//bit packed sint;
myStopMode.0 := bNo_Ramp_Stop;
myStopMode.1 := bFollowing_Error_Stop;

//34.001  AMC Stop Mode
//AMC StopMode(34.001)
WriteUserParameterSINT(00,34,001,myStopMode);
	
//41.007  AMC Following Error Window
//Set the following error window.
IF diFollowing_Error_Window < 0 THEN
	WriteUserParameterDINT(00,41,007,0);						//limit the value to no less then 
ELSE
	WriteUserParameterDINT(00,41,007,diFollowing_Error_Window);
END_IF

END_FUNCTION

// Drive/Application/Basic AMC Library/03 Commands/Stop/Stop_Motion
//Stops motion using the deceleration rate that you last used.
 

//Version 0.00.01
//Cannon Melville
FUNCTION Stop_Motion
VAR_INPUT
END_VAR 
VAR
END_VAR

(*	 
	Editing the code in this function may result in limited support. 	 
*)

(* NOTE
	Parameter 34.007  AMC Reference Select (Motion Commands)
	
	Value 	Disc 
	0 		Stop 
	1 		Position Abs 
	2 		Speed 
	3 		Cam 
	4 		EGB 
	5 		Home 
	6 		Position Rel 
	7 		Position Profile 
 
*)
 
//Stop command
//WriteUserParameterSINT(0,34,007,0);					//send a stop command
//Stop command - using the speed command set to zero speed.  
//This is becuase the AMC stop command does not like change in dec at the same time as a stop.
WriteUserParameterDINT(00,34,006,0);					//Set speed to 0	UU/ ms
WriteUserParameterINT(00,34,007,0);						//2= Start speed // change to 0 = stop // by Apikon Super Engineer
 

//35.010  AMC Cam Complete
WriteUserParameterBOOL(0,35,010,TRUE);				//Stop cam table

END_FUNCTION

// Drive/Application/Basic AMC Library/03 Commands/Stop/Stop_Motion_Decel
//Stops motion using a new deceleration rate.
//This block change the Deceleration rate.  Becuase there is a 4ms AMC update delay.  
//There is a possibility that the AMC will use the old deceleration rate for the first 4ms of the Deceleration.
//Also if the stop mode is set to no ramps then the AMC will not ramp down, instead it will stop immediately. See AMC_StopMode or parameter 34.001

//Version 0.00.01
//Cannon Melville
FUNCTION Stop_Motion_Decel
VAR_INPUT
	Deceleration 	: DINT;  //(38.002)  AMC Profile Deceleration  3 Decimal Places 
END_VAR 
VAR
END_VAR

(*	 
	Editing the code in this function may result in limited support. 	 
*)

(* NOTE
	Parameter 34.007  AMC Reference Select (Motion Commands)
	
	Value 	Disc 
	0 		Stop 
	1 		Position Abs 
	2 		Speed 
	3 		Cam 
	4 		EGB 
	5 		Home 
	6 		Position Rel 
	7 		Position Profile 
 
*)
 

//(38.002)  AMC Profile Deceleration  3 Decimal Places 
WriteUserParameterDINT(00,38,002,Deceleration);			//Set User Units Deceleration		UU/ ms^2

//Stop command
//WriteUserParameterSINT(0,34,007,0);					//send a stop command
//Stop command - using the speed command set to zero speed.  
//This is becuase the AMC stop command does not like change in dec at the same time as a stop.
WriteUserParameterDINT(00,34,006,0);					//Set speed to 0	UU/ ms
WriteUserParameterINT(00,34,007,2);						//2= Start speed
 

//35.010  AMC Cam Complete
WriteUserParameterBOOL(0,35,010,TRUE);					//Stop cam table

END_FUNCTION

// Drive/Application/Basic AMC Library/03 Commands/Index/Start_Index_ABS
 //Starts an index to a given position. 
 //Example: If the current position is 180 degrees and the distance passed to this function is 360 degrees then the motor will turn forward 180 degrees so that it stops at 360 degrees.
 //Example: If the current position is 360 degrees and the distance passed to this function is 360 degrees then the motor will not move.
 
 

//Version 0.00.02
//Cannon Melville
FUNCTION Start_Index_ABS
VAR_INPUT
	Acceleration 	: DINT;  //(38.001)  AMC Profile Acceleration  3 Decimal Places 
	Deceleration 	: DINT;  //(38.002)  AMC Profile Deceleration  3 Decimal Places 
	Velocity		: DINT;  //(38.003)  AMC Profile Max Speed  2 Decimal Places 
	Distance 		: DINT;  //(34.003)  AMC Position Reference  0 Decimal Places 
END_VAR

(*	 
	Editing the code in this function may result in limited support. 	 
*)

(* NOTE
	Parameter 34.007  AMC Reference Select (Motion Commands)
	
	Value 	Disc 
	0 		Stop 
	1 		Position Abs 
	2 		Speed 
	3 		Cam 
	4 		EGB 
	5 		Home 
	6 		Position Rel 
	7 		Position Profile 
 
*)
 
//needed to start the nexted index
IF ReadUserParameterSINT(0,34,007) > 1 THEN
	WriteUserParameterSINT(0,34,007,7);						//Profile mode	
END_IF


//Update profile generator
//(34.003)  AMC Position Reference  0 Decimal Places 
//(38.001)  AMC Profile Acceleration  3 Decimal Places 
//(38.002)  AMC Profile Deceleration  3 Decimal Places 
//(38.003)  AMC Profile Max Speed  2 Decimal Places 
WriteUserParameterDINT(00,34,003,Distance);				//Distance is abs from home or power up
WriteUserParameterDINT(00,38,001,Acceleration);			//Set User Units Acceleration		UU/ ms^2
WriteUserParameterDINT(00,38,002,Deceleration);			//Set User Units Deceleration		UU/ ms^2
WriteUserParameterDINT(00,38,003,ABS(Velocity));		//Set User Units Velocity			UU/ ms
	
//Wait 4ms so the the Drive can see that the values changed.
Wait_Time(T#4MS);
	
//start command
WriteUserParameterSINT(0,34,007,1);						//Start ABS Position.
	 
//Wait 4ms so the AMC motion flags can update.
//If you don't need the 4ms delay you can remove it to speed up the code.
Wait_Time(T#4MS);

END_FUNCTION

// Drive/Application/Basic AMC Library/03 Commands/Index/Start_Index_INC
//Starts an index from the current position plus the distance requested.
//This block has greater likelihood of having position Error versus Start_Index_REF over multiple indexes.

 //**Example #1: If the distance requested is 360 degrees, then each time you call this function the system will turn forward 360 degrees 
				//Plus or Minus the Movement Complete Window.
				
 //**Example #2: If the distance requested is -360 degrees, then each time you call this function the system will turn backwards 360 degrees 
				//Plus or Minus the Movement Complete Window.
				
 //**Example #3: If the System is moving and the current position is 180 degrees and the distance passed to this function is 360 degrees then 
				//the motor will turn forward 360 more degrees so that it stops at 540 degrees. ( Plus or Minus the Movement Complete Window.)
 
  
//Version 0.00.02
//Cannon Melville
FUNCTION Start_Index_INC
VAR_INPUT
	Acceleration 	: DINT;  //(38.001)  AMC Profile Acceleration  3 Decimal Places 
	Deceleration 	: DINT;  //(38.002)  AMC Profile Deceleration  3 Decimal Places 
	Velocity		: DINT;  //(38.003)  AMC Profile Max Speed  2 Decimal Places 
	Distance 		: DINT;  //(34.003)  AMC Position Reference  0 Decimal Places 
END_VAR
 

VAR
	diCurrentPosition: DINT;
END_VAR

(*	 
	Editing the code in this function may result in limited support. 	 
*)

(* NOTE
	Parameter 34.007  AMC Reference Select (Motion Commands)
	
	Value 	Disc 
	0 		Stop 
	1 		Position Abs 
	2 		Speed 
	3 		Cam 
	4 		EGB 
	5 		Home 
	6 		Position Rel 
	7 		Position Profile 
 
*)

//get position
diCurrentPosition := ReadUserParameterDINT(00,38,008);

//needed to start the nexted index
IF ReadUserParameterSINT(0,34,007) > 1 THEN
	WriteUserParameterSINT(0,34,007,7);						//Profile mode	
END_IF

//Update profile generator
//(34.003)  AMC Position Reference  0 Decimal Places 
//(38.001)  AMC Profile Acceleration  3 Decimal Places 
//(38.002)  AMC Profile Deceleration  3 Decimal Places 
//(38.003)  AMC Profile Max Speed  2 Decimal Places 
WriteUserParameterDINT(00,34,003,Distance + diCurrentPosition );	//Distance is abs from home or power up
WriteUserParameterDINT(00,38,001,Acceleration);			//Set User Units Acceleration		UU/ ms^2
WriteUserParameterDINT(00,38,002,Deceleration);			//Set User Units Deceleration		UU/ ms^2
WriteUserParameterDINT(00,38,003,ABS(Velocity));		//Set User Units Velocity			UU/ ms
	
//Wait 4ms so the the Drive can see that the values changed.
Wait_Time(T#4MS);
	
//start command
WriteUserParameterSINT(0,34,007,1);						//Start ABS Position.
	 
//Wait 4ms so the AMC motion flags can update.
//If you don't need the 4ms delay you can remove it to speed up the code.
Wait_Time(T#4MS);

END_FUNCTION

// Drive/Application/Basic AMC Library/03 Commands/Index/Start_Index_REF
//Starts an index from the last position target plus the distance requested.
//This block has less chance of position error over multiple indexs versus Start_Index_INC .

//**Example #1: If the distance requested is 360 degrees, then each time you call this function the system will turn forward 360 degrees.
//**Example #2: If the distance requested is -360 degrees, then each time you call this function the system will turn backwards 360 degrees.
//**Example #3: If the system was originally given a target position of 360 degrees, the system is now moving, the current position is 180 degrees, 
			//and the distance passed to this function is 360 degrees then the motor will turn forward 540 more degrees so that it stops at 720 degrees. 

  

//Version 0.00.03
//Cannon Melville
FUNCTION Start_Index_REF
VAR_INPUT
	Acceleration 	: DINT;  //(38.001)  AMC Profile Acceleration  3 Decimal Places 
	Deceleration 	: DINT;  //(38.002)  AMC Profile Deceleration  3 Decimal Places 
	Velocity		: DINT;  //(38.003)  AMC Profile Max Speed  2 Decimal Places 
	Distance 		: DINT;  //(34.003)  AMC Position Reference  0 Decimal Places 
END_VAR

VAR
	diCurrentPosition: DINT;
END_VAR

(*	 
	Editing the code in this function may result in limited support. 	 
*)

(* NOTE
	Parameter 34.007  AMC Reference Select (Motion Commands)
	
	Value 	Disc 
	0 		Stop 
	1 		Position Abs 
	2 		Speed 
	3 		Cam 
	4 		EGB 
	5 		Home 
	6 		Position Rel 
	7 		Position Profile 
 
*)
 

//get position
diCurrentPosition := ReadUserParameterDINT(00,38,006);


//needed to start the nexted index
IF ReadUserParameterSINT(0,34,007) > 1 THEN
	WriteUserParameterSINT(0,34,007,7);						//Profile mode	
END_IF

//Update profile generator
//(34.003)  AMC Position Reference  0 Decimal Places 
//(38.001)  AMC Profile Acceleration  3 Decimal Places 
//(38.002)  AMC Profile Deceleration  3 Decimal Places 
//(38.003)  AMC Profile Max Speed  2 Decimal Places 
WriteUserParameterDINT(00,34,003,Distance + diCurrentPosition );	//Distance is abs from home or power up
WriteUserParameterDINT(00,38,001,Acceleration);			//Set User Units Acceleration		UU/ ms^2
WriteUserParameterDINT(00,38,002,Deceleration);			//Set User Units Deceleration		UU/ ms^2
WriteUserParameterDINT(00,38,003,ABS(Velocity));		//Set User Units Velocity			UU/ ms
	
//Wait 4ms so the the Drive can see that the values changed.
Wait_Time(T#4MS);
	
//start command
WriteUserParameterSINT(0,34,007,1);						//Start ABS Position.
	 
//Wait 4ms so the AMC motion flags can update.
//If you don't need the 4ms delay you can remove it to speed up the code.
Wait_Time(T#4MS);

END_FUNCTION

// Drive/Application/Basic AMC Library/03 Commands/Jog/Start_Jog_Minus
//Starts a speed reverse command.


//Version 0.00.01
//Cannon Melville 
 FUNCTION Start_Jog_Minus
VAR_INPUT
	Acceleration 	: DINT;  //(38.001)  AMC Profile Acceleration  3 Decimal Places 
	Deceleration 	: DINT;  //(38.002)  AMC Profile Deceleration  3 Decimal Places 
	Velocity		: DINT;  //(38.003) & (34.006) AMC Profile Max Speed  2 Decimal Places 
END_VAR 
VAR

END_VAR

(*	 
	Editing the code in this function may result in limited support. 	 
*)

(* NOTE
	Parameter 34.007  AMC Reference Select (Motion Commands)
	
	Value 	Disc 
	0 		Stop 
	1 		Position Abs 
	2 		Speed 
	3 		Cam 
	4 		EGB 
	5 		Home 
	6 		Position Rel 
	7 		Position Profile 
 
*)

//needed to start the nexted index
//WriteUserParameterSINT(0,34,007,7);						//Profile mode

//Update profile generator
//(34.006)  AMC Jog Speed  2 Decimal Places 
//(38.001)  AMC Profile Acceleration  3 Decimal Places 
//(38.002)  AMC Profile Deceleration  3 Decimal Places 
//(38.003)  AMC Profile Max Speed  2 Decimal Places 
WriteUserParameterDINT(00,38,001,Acceleration);			//Set User Units Acceleration		UU/ ms^2
WriteUserParameterDINT(00,38,002,Deceleration);			//Set User Units Deceleration		UU/ ms^2
WriteUserParameterDINT(00,38,003,ABS(Velocity));		//Set User Units Velocity			UU/ ms
WriteUserParameterDINT(00,34,006,-Velocity);			//Set User Units Velocity			UU/ ms
	
//Wait 4ms so the the Drive can see that the values changed.
Wait_Time(T#4MS);
	
//Start the speed
WriteUserParameterINT(00,34,007,2);						//2= Start speed

END_FUNCTION

// Drive/Application/Basic AMC Library/03 Commands/Jog/Start_Jog_Plus
//Starts a speed forward command.


//Version 0.00.02
//Cannon Melville 
FUNCTION Start_Jog_Plus
VAR_INPUT
	Acceleration 	: DINT;  //(38.001)  AMC Profile Acceleration  3 Decimal Places 
	Deceleration 	: DINT;  //(38.002)  AMC Profile Deceleration  3 Decimal Places 
	Velocity		: DINT;  //(38.003) & (34.006) AMC Profile Max Speed  2 Decimal Places 
END_VAR 
VAR

END_VAR

(*	 
	Editing the code in this function may result in limited support. 	 
*)

(* NOTE
	Parameter 34.007  AMC Reference Select (Motion Commands)
	
	Value 	Disc 
	0 		Stop 
	1 		Position Abs 
	2 		Speed 
	3 		Cam 
	4 		EGB 
	5 		Home 
	6 		Position Rel 
	7 		Position Profile 
 
*)

//needed to start the nexted index
//WriteUserParameterSINT(0,34,007,7);						//Profile mode

//Update profile generator
//(34.006)  AMC Jog Speed  2 Decimal Places 
//(38.001)  AMC Profile Acceleration  3 Decimal Places 
//(38.002)  AMC Profile Deceleration  3 Decimal Places 
//(38.003)  AMC Profile Max Speed  2 Decimal Places 
WriteUserParameterDINT(00,38,001,Acceleration);			//Set User Units Acceleration		UU/ ms^2
WriteUserParameterDINT(00,38,002,Deceleration);			//Set User Units Deceleration		UU/ ms^2
WriteUserParameterDINT(00,38,003,ABS(Velocity));		//Set User Units Velocity			UU/ ms
WriteUserParameterDINT(00,34,006,Velocity);				//Set User Units Velocity			UU/ ms
	
//Wait 4ms so the the Drive can see that the values changed.
Wait_Time(T#4MS);
	
//Start the Speed
WriteUserParameterINT(00,34,007,2);						//2= Start speed

END_FUNCTION

// Drive/Application/Basic AMC Library/03 Commands/EGB/Start_Gearing
(*
---- RIGID MODE = FALSE ----
If AMC EGB Enable Rigid Mode (37.001) = 0, then the system attempts to match the speed of the slave with the speed of the master. 
The speed at the output of the profile generator can only change within the acceleration/deceleration constraints. 
This function sets up the profile generator (i.e. AMC Profile Acceleration (38.001), AMC Profile Deceleration (38.002) and AMC Profile Maximum Speed (38.003)). 
Once the difference between the speed at the input and output of the profile generator is less than or equal to
AMC EGB Locking Speed Band (37.004), the profile generator is disabled.  At this point the sytem is locked. 


---- RIGID MODE = True ----
If AMC EGB Enable Rigid Mode (37.001) = 1 the system attempts to match the speed and position of the slave before changing to the locked state. 
The profile generator output will exceed the profile generator input speed to make up the position lost during acceleration. 
The system only changes to the locked state when the speed difference between the input and output of the profile generator is within the AMC EGB 
Locking Speed Band (37.004), and the difference between the input and output position is within the AMC EGB Locking Position Band (37.005).
 
*) 
//Version 0.00.02
//Cannon Melville 
 FUNCTION Start_Gearing
VAR_INPUT
	Acceleration 	: DINT;  //(38.001)  AMC Profile Acceleration  3 Decimal Places 
	Deceleration 	: DINT;  //(38.002)  AMC Profile Deceleration  3 Decimal Places 
	MaxVelocity		: DINT;  //(38.003)  AMC Profile Max Speed  2 Decimal Places 
	
	EGB_RigidMode				: BOOL; //(37.001)  AMC EGB Enable Rigid Lock
	EGB_RatioNumerator			: DINT;	//(37.002)  AMC EGB Ratio Numerator Default = 1000
	EGB_RatioDenominator		: DINT;	//(37.003)  AMC EGB Ratio Denominator Default = 1000
	EGB_Locking_SpeedBand		: DINT;	//(37.004)  AMC EGB Locking Speed Band, 2 decimal places.
	EGB_Locking_PositionBand	: DINT;	//(37.005)  AMC EGB Locking Position Band, 0 decimal places.  
	
END_VAR 
VAR

END_VAR

(*	 
	Editing the code in this function may result in limited support. 	 
*)

(* NOTE
	Parameter 34.007  AMC Reference Select (Motion Commands)
	
	Value 	Disc 
	0 		Stop 
	1 		Position Abs 
	2 		Speed 
	3 		Cam 
	4 		EGB 
	5 		Home 
	6 		Position Rel 
	7 		Position Profile 
 
*)

//needed to start the nexted index
//WriteUserParameterSINT(0,34,007,7);						//Profile mode

//Update profile generator
//(34.006)  AMC Jog Speed  2 Decimal Places 
//(38.001)  AMC Profile Acceleration  3 Decimal Places 
//(38.002)  AMC Profile Deceleration  3 Decimal Places 
//(38.003)  AMC Profile Max Speed  2 Decimal Places 
WriteUserParameterDINT(00,38,001,Acceleration);			//Set User Units Acceleration		UU/ ms^2
WriteUserParameterDINT(00,38,002,Deceleration);			//Set User Units Deceleration		UU/ ms^2
WriteUserParameterDINT(00,38,003,ABS(MaxVelocity));		//Set User Units Velocity			UU/ ms 

//(37.001)  AMC EGB Enable Rigid Lock
//(37.001)  AMC EGB Enable Rigid Lock
//(37.002)  AMC EGB Ratio Numerator 
//(37.003)  AMC EGB Ratio Denominator
//(37.004)  AMC EGB Locking Speed Band
//(37.005)  AMC EGB Locking Position Band
WriteUserParameterBOOL(00,37,001,EGB_RigidMode);			//Enable Rigid mode
WriteUserParameterDINT(00,37,002,EGB_RatioNumerator);		//
WriteUserParameterDINT(00,37,003,EGB_RatioDenominator);		//
WriteUserParameterDINT(00,37,004,EGB_Locking_SpeedBand);	//2 decimal places.
WriteUserParameterDINT(00,37,005,EGB_Locking_PositionBand);	// 
	
//Wait 4ms so the the Drive can see that the values changed.
Wait_Time(T#4MS);
	
//Start the Speed
WriteUserParameterINT(00,34,007,4);						//4= Start Gearing

END_FUNCTION

// Drive/Application/Basic AMC Library/10 Other/ScaleValue_DI
 
//This is good for units manipulation
//Compatible with M400, M700, MCI200, MCI210
//Verison 0.02.00
//Cannon Melville  
FUNCTION ScaleValue_DI  
 
VAR_INPUT
	diNewInputValue	: DINT := 0;				//input value
	diMaxInputValue	: DINT := 0;				//input value
	diMinInputValue	: DINT := 0;				//input value
	
	DIMaxOuputValue	: DINT := 0;				//input value
	DIMinOuputValue	: DINT := 0;				//input value
		
	// If true the output value will not exceed the max and min.
	bLimmitOutput	: BOOL := FALSE;
	
END_VAR

VAR_OUTPUT 
	
	diScaledValue	: DINT;
	bError 			: BOOL;
END_VAR

VAR 
	diTemp : DINT; 
	 
END_VAR

(*	LEVEL NA SUPPORT
	This block is Not supported  	 
*)


(*
	This block scales the input value to an output value.
	All inputs need to be setup.
*)
 
diTemp := diMaxInputValue - diMinInputValue;

IF diTemp = 0   THEN
	diScaledValue 	:= 0;				//Error can't / by 0
	bError 			:= TRUE;
ELSE
	
	
	//Limmit output if needed
	IF bLimmitOutput = TRUE THEN		
		// limit to max value
		IF diNewInputValue > diMaxInputValue THEN
			diNewInputValue := diMaxInputValue;
		END_IF
		// Limit to min value
		IF diNewInputValue <  diMinInputValue THEN 
			diNewInputValue := diMinInputValue;
		END_IF 				
	END_IF


	//Scale the Value
	diScaledValue := ( (diNewInputValue - diMinInputValue) * (diMaxOuputValue - diMinOuputValue) ) / ( diTemp )   +  diMinOuputValue ;  
  
	(*Old way
	 //Limmit output if needed
	IF bLimmitOutput = TRUE THEN
		IF diScaledValue > diMaxOuputValue THEN
			diScaledValue := diMaxOuputValue;
		END_IF
		IF diScaledValue < diMinOuputValue THEN 
			diScaledValue := diMinOuputValue;
		END_IF
	END_IF
	*)
	
	//update the output value
	//ScaleValue_DI :=	diScaledValue; 	
END_IF

END_FUNCTION

// Drive/Application/Program/Freewheeling
PROGRAM Freewheeling
VAR
	ALWAYS_ON: BOOL := TRUE;
	Start_ABS_Move: BOOL := FALSE;
	FinalDistance: DINT := 0;
	SelectDistance: BOOL := FALSE;
	SecondDistance: BOOL := FALSE;
	FWDPos_Reached: BOOL;
	REVPos_Reached: BOOL;
	PBPress_States: WORD := 0;
	StartHome: BOOL := FALSE;
	FWD_Wait_Time: TON;
	REV_Wait_Time: TON;
	FWD_Idle_Time: TIME;
	REV_Idle_Time: TIME;
	FWD_Waiting_Time: TIME;
	REV_Waiting_Time: TIME;
	PercentagePos: DINT;
	OpenGate: BOOL := FALSE;
	Stop_ABS_Move: BOOL := FALSE;
	StopMotionSelected: BOOL := FALSE;
	
	//SCALE VALUE FOR PERCENTAGE	
	ScaleError: BOOL := FALSE;

	AccelIndex1: DINT;
	DecelIndex1: DINT;
	VelocityIndex1: INT := 2000;
	StartJog: BOOL := FALSE;
	StartJogPlus: BOOL := FALSE;
	StartJogMinus: BOOL := false;
	cut_pule: BOOL := FALSE;
	TP_0: TP;
	Counter_Value: INT;
	COUNTER_MATERIAL: CTU;
END_VAR
VAR_OUTPUT
	cut_pulse: BOOL := FALSE;
END_VAR
VAR // added by the converter: edge detectors and wires of the graphical bodies
    _rt1, _rt2, _rt3, _rt4 : R_TRIG;
    _w1, _w2, _w3 : BOOL;
    _ft1, _ft2 : F_TRIG;
END_VAR

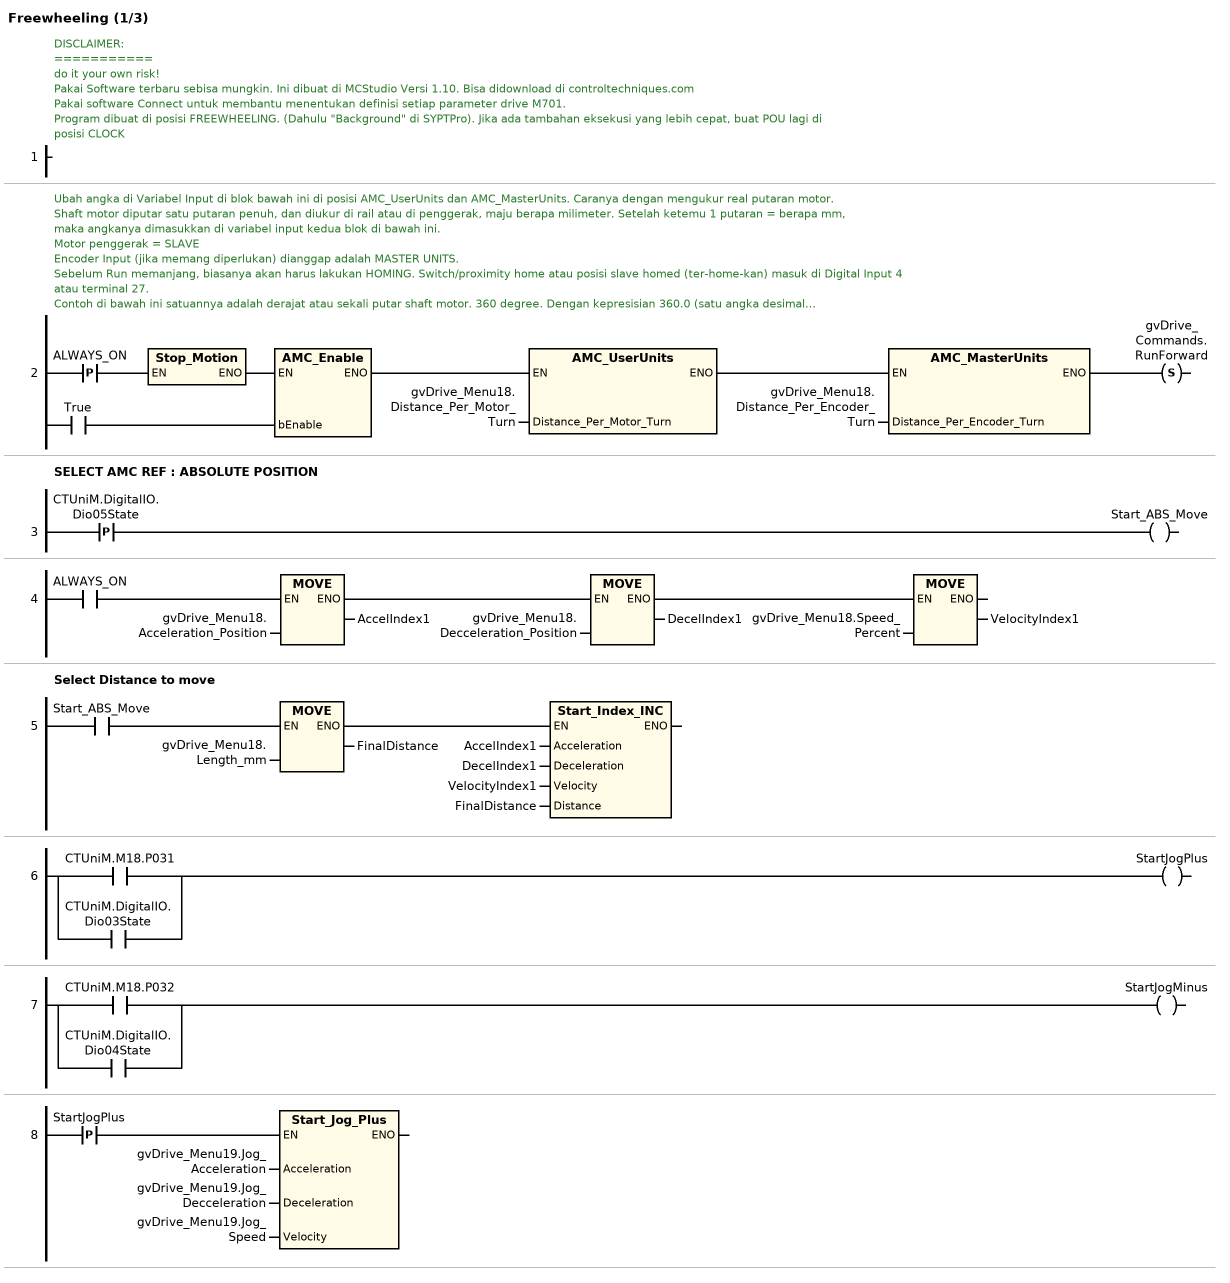
// NETWORK 1
// DISCLAIMER:
// 	===========
// 	do it your own risk!
//
// 	Pakai Software terbaru sebisa mungkin. Ini dibuat di MCStudio Versi 1.10. Bisa didownload di controltechniques.com
// 	Pakai software Connect untuk membantu menentukan definisi setiap parameter drive M701.
//
// Program dibuat di posisi FREEWHEELING. (Dahulu "Background" di SYPTPro). Jika ada tambahan eksekusi yang lebih cepat, buat POU lagi di
// posisi CLOCK

// NETWORK 2
// Ubah angka di Variabel Input di blok bawah ini di posisi AMC_UserUnits dan AMC_MasterUnits. Caranya dengan mengukur real putaran motor.
// Shaft motor diputar satu putaran penuh, dan diukur di rail atau di penggerak, maju berapa milimeter. Setelah ketemu 1 putaran = berapa mm,
// maka angkanya dimasukkan di variabel input kedua blok di bawah ini.
//
// Motor penggerak = SLAVE
// Encoder Input (jika memang diperlukan) dianggap adalah MASTER UNITS.
//
// Sebelum Run memanjang, biasanya akan harus lakukan HOMING. Switch/proximity home atau posisi slave homed (ter-home-kan) masuk di Digital Input 4
// atau terminal 27.
//
// Contoh di bawah ini satuannya adalah derajat atau sekali putar shaft motor. 360 degree. Dengan kepresisian 360.0 (satu angka desimal)
// Makanya User Unitnya tertulis 3600 alias 360.0. Pilihan lain disesuaikan dengan aplikasi di lapangan.
_rt1(CLK := ALWAYS_ON);
_w1 := _rt1.Q;
IF _w1 THEN Stop_Motion(); END_IF
IF _w1 THEN AMC_Enable(bEnable := True); END_IF
IF _w1 THEN AMC_UserUnits(Distance_Per_Motor_Turn := gvDrive_Menu18.Distance_Per_Motor_Turn); END_IF
IF _w1 THEN AMC_MasterUnits(Distance_Per_Encoder_Turn := gvDrive_Menu18.Distance_Per_Encoder_Turn); END_IF
gvDrive_Commands.RunForward S= _w1;

// NETWORK 3: SELECT AMC REF : ABSOLUTE POSITION
_rt2(CLK := CTUniM.DigitalIO.Dio05State);
Start_ABS_Move := _rt2.Q;

// NETWORK 4
_w2 := ALWAYS_ON;
IF _w2 THEN AccelIndex1 := gvDrive_Menu18.Acceleration_Position; END_IF
IF _w2 THEN DecelIndex1 := gvDrive_Menu18.Decceleration_Position; END_IF
IF _w2 THEN VelocityIndex1 := gvDrive_Menu18.Speed_Percent; END_IF

// NETWORK 5: Select Distance to move
_w3 := Start_ABS_Move;
IF _w3 THEN FinalDistance := gvDrive_Menu18.Length_mm; END_IF
IF _w3 THEN
    Start_Index_INC(Acceleration := AccelIndex1, Deceleration := DecelIndex1, Velocity := VelocityIndex1, Distance := FinalDistance);
END_IF

// NETWORK 6
StartJogPlus := CTUniM.M18.P031 OR CTUniM.DigitalIO.Dio03State;

// NETWORK 7
StartJogMinus := CTUniM.M18.P032 OR CTUniM.DigitalIO.Dio04State;

// NETWORK 8
_rt3(CLK := StartJogPlus);
IF _rt3.Q THEN
    Start_Jog_Plus(Acceleration := gvDrive_Menu19.Jog_Acceleration, Deceleration := gvDrive_Menu19.Jog_Decceleration, Velocity := gvDrive_Menu19.Jog_Speed);
END_IF

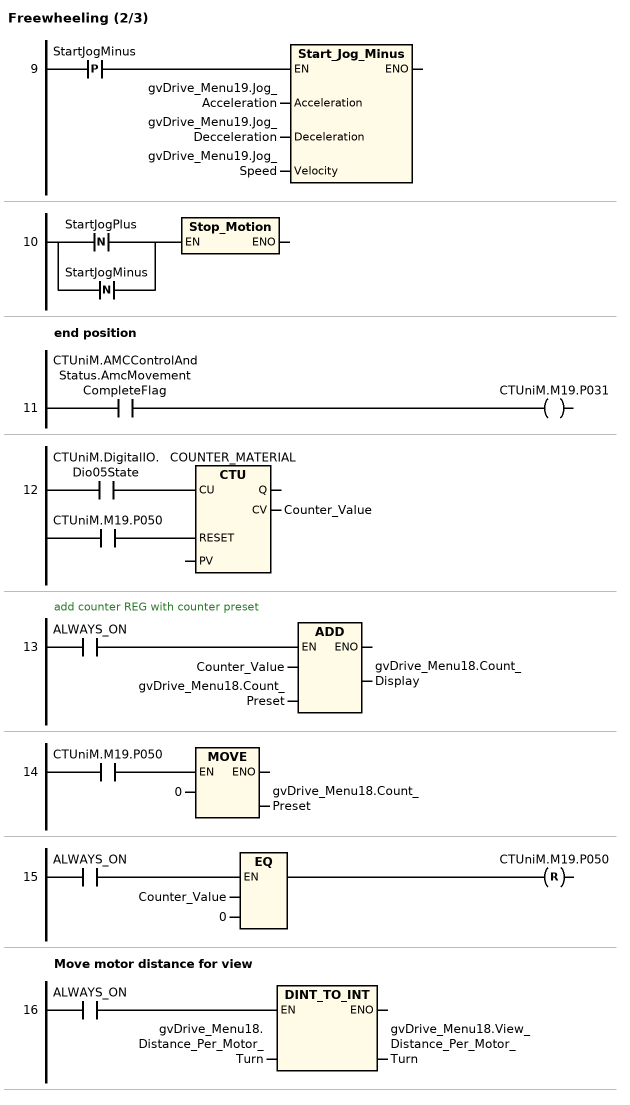
// NETWORK 9
_rt4(CLK := StartJogMinus);
IF _rt4.Q THEN
    Start_Jog_Minus(Acceleration := gvDrive_Menu19.Jog_Acceleration, Deceleration := gvDrive_Menu19.Jog_Decceleration, Velocity := gvDrive_Menu19.Jog_Speed);
END_IF

// NETWORK 10
_ft1(CLK := StartJogPlus);
_ft2(CLK := StartJogMinus);
IF _ft1.Q OR _ft2.Q THEN Stop_Motion(); END_IF

// NETWORK 11: end position
CTUniM.M19.P031 := CTUniM.AMCControlAndStatus.AmcMovementCompleteFlag;

// NETWORK 12
COUNTER_MATERIAL(CU := CTUniM.DigitalIO.Dio05State, RESET := CTUniM.M19.P050, CV => Counter_Value); // CTU

// NETWORK 13
// add counter REG with counter preset
IF ALWAYS_ON THEN gvDrive_Menu18.Count_Display := Counter_Value + gvDrive_Menu18.Count_Preset; END_IF

// NETWORK 14
IF CTUniM.M19.P050 THEN gvDrive_Menu18.Count_Preset := 0; END_IF

// NETWORK 15
CTUniM.M19.P050 R= ALWAYS_ON AND Counter_Value = 0;

// NETWORK 16: Move motor distance for view
IF ALWAYS_ON THEN
    gvDrive_Menu18.View_Distance_Per_Motor_Turn := DINT_TO_INT(gvDrive_Menu18.Distance_Per_Motor_Turn);
END_IF

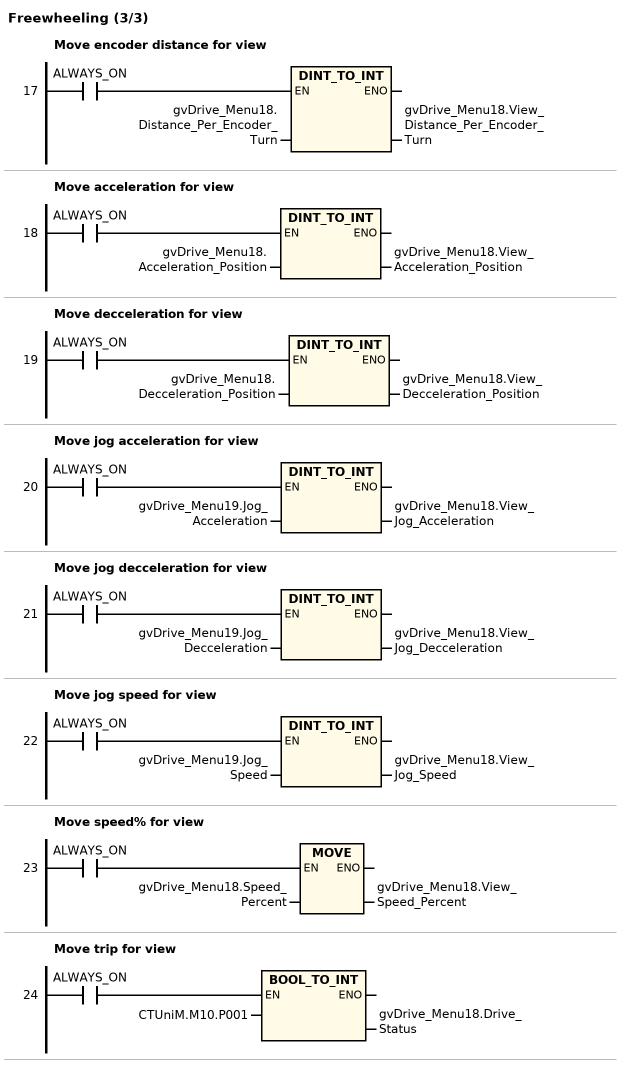
// NETWORK 17: Move encoder distance for view
IF ALWAYS_ON THEN
    gvDrive_Menu18.View_Distance_Per_Encoder_Turn := DINT_TO_INT(gvDrive_Menu18.Distance_Per_Encoder_Turn);
END_IF

// NETWORK 18: Move acceleration for view
IF ALWAYS_ON THEN
    gvDrive_Menu18.View_Acceleration_Position := DINT_TO_INT(gvDrive_Menu18.Acceleration_Position);
END_IF

// NETWORK 19: Move decceleration for view
IF ALWAYS_ON THEN
    gvDrive_Menu18.View_Decceleration_Position := DINT_TO_INT(gvDrive_Menu18.Decceleration_Position);
END_IF

// NETWORK 20: Move jog acceleration for view
IF ALWAYS_ON THEN gvDrive_Menu18.View_Jog_Acceleration := DINT_TO_INT(gvDrive_Menu19.Jog_Acceleration); END_IF

// NETWORK 21: Move jog decceleration for view
IF ALWAYS_ON THEN gvDrive_Menu18.View_Jog_Decceleration := DINT_TO_INT(gvDrive_Menu19.Jog_Decceleration); END_IF

// NETWORK 22: Move jog speed for view
IF ALWAYS_ON THEN gvDrive_Menu18.View_Jog_Speed := DINT_TO_INT(gvDrive_Menu19.Jog_Speed); END_IF

// NETWORK 23: Move speed% for view
IF ALWAYS_ON THEN gvDrive_Menu18.View_Speed_Percent := gvDrive_Menu18.Speed_Percent; END_IF

// NETWORK 24: Move trip for view
IF ALWAYS_ON THEN gvDrive_Menu18.Drive_Status := BOOL_TO_INT(CTUniM.M10.P001); END_IF

END_PROGRAM

// Drive/Application/Basic AMC Library/03 Commands/Home/Set_Position
(*
	This home command set the position without moving the system.  The system must be stopped for this block to work.
	
	This function does 3 things.
	1. Test to see if the drive is Active 
	2. Run homing mode
	3. Test for error 
 
 
	Note : This function needs to be able to toggle the value in parameter 40.012.  If a digital input is map to Parameter 40.012
	this function will not work.
*)
 


FUNCTION Set_Position 
VAR_INPUT
	SetPosition : DINT;  		//This is the position the system is at right now.
	
END_VAR
VAR_OUTPUT
	xError		:BOOL;			//Drive must be enabled and stopped for this block to work.	Also there is a test to see if the home flag 	
END_VAR
VAR
END_VAR

(*	 
	Editing the code in this function may result in limited support. 	 
*)


//Test for Errors.	
xError := FALSE;
IF ReadUserParameterBool(00,10,002) = FALSE THEN						//Drive needs to be Active
	xError := TRUE;
	RETURN;
END_IF	
IF ReadUserParameterBool(00,34,007) > 0 THEN							//Drive must have a stop command
	xError := TRUE;
	RETURN;
END_IF

	//clear home offset
	WriteUserParameterDINT(00,33,003,0);					//clear position offset;
	Wait_Time(T#30MS);										//wait 30 ms	
	

	//-----------------------------------------setup------------------------------------------\\
	
	//Menu 40
	//WriteUserParameterBOOL(00,40,001,0);					//Home Direction	
	WriteUserParameterSINT(00,40,002,0);					//Home mode 1
	WriteUserParameterDINT(00,40,003,0);					//Home max speed
	WriteUserParameterDINT(00,40,004,SetPosition);			//Home Position
	  
	WriteUserParameterDINT(00,40,007,0);					//Home Offset Position 
 
		
	//40.011  AMC Home On Freeze
	//40.012  AMC Home Switch	
	WriteUserParameterBOOL(00,40,011,FALSE);				//dont use the freeze
	WriteUserParameterBOOL(00,40,014,FALSE);				//Stop now limit.  Turn this off so the motion can run.
				
	//40.015  AMC Home Positive Limit Selector
	//40.016  AMC Home Negative Limit Selector
	WriteUserParameterLREAL(00,40,018,0);					//Torque level
	WriteUserParameterLREAL(00,40,019,0);					//Torque Delay Time		
	
	//-----------------------------------------home the Drive------------------------------------------\\
	WriteUserParameterBOOL(00,40,012,0);					//Clear Home Switch
	Wait_Time(T#30MS);										//wait 30 ms
 
	WriteUserParameterSINT(00,34,007,5);					//Start home

	Wait_Time(T#30MS);										//wait 30 ms
	WriteUserParameterBOOL(00,40,012,1);					//Set Home Switch												
	
	Wait_Time(T#30MS);										//wait 30 ms														
	IF NOT ReadUserParameterBOOL(0,40,005) THEN				//did the home get done.
		xError	:= TRUE;									//error if it did not work.
	END_IF

END_FUNCTION

// Drive/Application/Basic AMC Library/03 Commands/Home/Start_Homing_To_Input_4
//Starts a home command that completes after input 4 turns on.
 

//Version 0.00.03
//Cannon Melville 
FUNCTION Start_Homing_To_Input_4
VAR_INPUT 
	Acceleration 		: DINT;
	Deceleration 		: DINT;
	Velocity			: DINT; 
	MaxAllowedMove		: DINT;	 // The max distance the home will run. 0 = disabled
	
	bHomeNegativeDirection	: BOOL;  // Home in the Negative Direction
	
	HomeCompleteWindow	: DINT;	 // This is used with the home complete flag
	HomeSwitchPosition 	: DINT;  // This is the position of the Home Switch or the homed position.

	OffsetSpeed			: DINT;  // This is the speed the system will move as the position reset, after the home switch is found.
	OffsetPosition 		: DINT;  // This is the offset position from the home switch to go to after the home is done.
	
	
	
END_VAR 
VAR

END_VAR

(*	 
	Editing the code in this function may result in limited support. 	 
*)

(* NOTE
	Parameter 34.007  AMC Reference Select (Motion Commands)
	
	Value 	Disc 
	0 		Stop 
	1 		Position Abs 
	2 		Speed 
	3 		Cam 
	4 		EGB 
	5 		Home 
	6 		Position Rel 
	7 		Position Profile 
 
*)
 									//wait 30 ms	
	


//Update profile generator 
//38.001  AMC Profile Acceleration
//38.002  AMC Profile Deceleration
//38.003  AMC Profile Maximum Speed
//40.003  AMC Home Maximum Speed
WriteUserParameterDINT(00,38,001,Acceleration);				//Set User Units Acceleration		UU/ ms^2
WriteUserParameterDINT(00,38,002,Deceleration);				//Set User Units Deceleration		UU/ ms^2
WriteUserParameterDINT(00,38,003,ABS(Velocity));			//Set User Units Velocity			UU/ ms
	

//menu 3
//03.100  F1 Freeze Trigger Source
//03.102  F1 Freeze Position Source
WriteUserParameterSINT(00,03,100,0);						//Use digital input 4
WriteUserParameterSINT(00,03,102,0);						//Use P1		
	
//menu 8
WriteUserParameterLREAL(00,08,024,0); 						//map input 4 to nothing	
	
//menu 33 Slave freeze Select
//33.007  AMC Slave Freeze Select
WriteUserParameterBOOL(00,33,007,0);						//Select Freeze 1 input as home switch
		
//Menu 40
//40.001  AMC Home Direction
//40.002  AMC Home Mode
//40.003  AMC Home Maximum Speed
//40.004  AMC Home Position
WriteUserParameterBOOL(00,40,001,bHomeNegativeDirection);	//Home Direction	
WriteUserParameterSINT(00,40,002,1);						//Home mode 1
WriteUserParameterDINT(00,40,003,Velocity);					//Set User Units Velocity			UU/ms
WriteUserParameterDINT(00,40,004,HomeSwitchPosition);		//Home  Switch Position
	 
//40.006  AMC Home Offset Maximum Speed
//40.007  AMC Home Offset Position
WriteUserParameterDINT(00,40,006,OffsetSpeed);				//Home offset Speed
WriteUserParameterDINT(00,40,007,OffsetPosition);			//Home offset Position 
	
//40.009  AMC Home Maximum Allowed Move
//40.010  AMC Home Complete Window
WriteUserParameterDINT(00,40,009,MaxAllowedMove);			//Home Max Allowed Move
WriteUserParameterDINT(00,40,010,HomeCompleteWindow);		//Home Home Complete Window
	
//40.011  AMC Home On Freeze
//40.012  AMC Home Switch	
WriteUserParameterBOOL(00,40,011,FALSE);					//dont use the freeze
WriteUserParameterBOOL(00,40,014,FALSE);					//Stop now limit.  Turn this off so the motion can run.
		
//40.013  AMC Home Positive Limit
//40.014  AMC Home Negative Limit
WriteUserParameterBOOL(00,40,015,FALSE);					//Disable the torque limit pos
WriteUserParameterBOOL(00,40,016,FALSE);					//Disable the torque limit neg
		
//40.015  AMC Home Positive Limit Selector
//40.016  AMC Home Negative Limit Selector
WriteUserParameterLREAL(00,40,018,0);						//Torque level
WriteUserParameterLREAL(00,40,019,0);						//Torque Delay Time
 

//Wait 4ms so the the Drive can see that the values changed.
Wait_Time(T#4MS);

	 
//Start the Homing using the trigger command and the normal command 
//34.007  AMC Reference Select
WriteUserParameterINT(00,34,007,5);							//5 = Start Homing

END_FUNCTION

// Drive/Application/Basic AMC Library/03 Commands/Home/Start_Homing_To_Input_4_Then_Marker
//Starts a home command that completes after input 4 turns on and then a marker or zero


//Version 0.00.03
//Cannon Melville 
FUNCTION Start_Homing_To_Input_4_Then_Marker
VAR_INPUT 
	Acceleration 		: DINT;
	Deceleration 		: DINT;
	Velocity			: DINT; 
	MaxAllowedMove		: DINT;	 // The max distance the home will run. 0 = disabled
	
	bHomeNegativeDirection	: BOOL;  // Home in the Negative Direction
	
	HomeCompleteWindow	: DINT;	 // This is used with the home complete flag
	HomeCompletePosition: DINT;  // This is the position of the homed after the torque value is reached.

	OffsetSpeed			: DINT;  // This is the speed the system will move as the position reset, after the home switch is found.
	OffsetPosition 		: DINT;  // This is the offset position from the home switch to go to after the home is done.
	
	bBackOffAfterInput4	: BOOL;  //after the torque Treshold and Torque Time Delay is met, Then reverse the directoin.

	
	
END_VAR 
VAR
 
END_VAR

(*	 
	Editing the code in this function may result in limited support. 	 
*)

(* NOTE
	Parameter 34.007  AMC Reference Select (Motion Commands)
	
	Value 	Disc 
	0 		Stop 
	1 		Position Abs 
	2 		Speed 
	3 		Cam 
	4 		EGB 
	5 		Home 
	6 		Position Rel 
	7 		Position Profile 
 
*)

//clear home offset
WriteUserParameterDINT(00,33,003,0);		//clear position offset;  This needs to happen with FW 1.15 and older.  I don't know if the newer FW need this.
Wait_Time(T#30MS);										//wait 30 ms	

  
//Update profile generator 
//38.001  AMC Profile Acceleration
//38.002  AMC Profile Deceleration
//38.003  AMC Profile Maximum Speed
//40.003  AMC Home Maximum Speed
WriteUserParameterDINT(00,38,001,Acceleration);				//Set User Units Acceleration		UU/ ms^2
WriteUserParameterDINT(00,38,002,Deceleration);				//Set User Units Deceleration		UU/ ms^2
WriteUserParameterDINT(00,38,003,ABS(Velocity));			//Set User Units Velocity			UU/ ms
	

//menu 3
//03.100  F1 Freeze Trigger Source
//03.102  F1 Freeze Position Source
IF ReadUserParameterSINT(00,03,038) = 0 OR ReadUserParameterSINT(00,03,038) = 3 THEN				//P1 Device Type(03.038) = AB Encoder then use marker else use 0 position Crossing
	WriteUserParameterSINT(00,03,100,2);					//Use digital P1 Marker
ELSE
	WriteUserParameterSINT(00,03,100,5);					//Use digital P1 Zero Position	
END_IF
WriteUserParameterSINT(00,03,102,0);						//Use P1		
	

//menu 33 Slave freeze Select
//33.007  AMC Slave Freeze Select
WriteUserParameterBOOL(00,33,007,0);						//Select Freeze 1 input as home switch
	
	
		
//Menu 40

//Direction settings
IF bHomeNegativeDirection THEN								//---- Negative direction ----	

	//map drive input 4 to home parameter
	WriteUserParameterLREAL(00,08,024,40.014); //map input 4 to the home	

	//40.002  AMC Home Mode
	WriteUserParameterSINT(00,40,002,3);					//Home mode 3  (i'm using this mode to do the neg direction)
 
	//40.001  AMC Home Direction after torque is met
	IF bBackOffAfterInput4 THEN
		WriteUserParameterBOOL(00,40,001,FALSE);					//Home Direction 
	ELSE
		WriteUserParameterBOOL(00,40,001,TRUE);				//Home Direction 
	END_IF
	
ELSE	
 
	//map drive input 4 to home parameter
	WriteUserParameterLREAL(00,08,024,40.013); //map input 4 to the home	
 											//---- Positive Direction ----
	//40.002  AMC Home Mode
	WriteUserParameterSINT(00,40,002,2);					//Home mode 2(i'm using this mode to do the Pos direction)
 
	//40.001  AMC Home Direction after torque is met
	IF bBackOffAfterInput4 THEN
		WriteUserParameterBOOL(00,40,001,TRUE);					//Home Direction 
	ELSE
		WriteUserParameterBOOL(00,40,001,FALSE);				//Home Direction 
	END_IF
	
END_IF


//reset the drive
WriteUserParameterUSINT(00,10,038,100); //command reset the drive //use new settings
Wait_Time(T#100MS); //delay 100ms 
WriteUserParameterUSINT(00,10,038,0); // command clear the reset



//40.001  AMC Home Direction
//40.003  AMC Home Maximum Speed
//40.004  AMC Home Position
WriteUserParameterDINT(00,40,003,Velocity);					//Set User Units Velocity			UU/ms
WriteUserParameterDINT(00,40,004,HomeCompletePosition);		//Home  Switch Position
	 
//40.006  AMC Home Offset Maximum Speed
//40.007  AMC Home Offset Position
WriteUserParameterDINT(00,40,006,OffsetSpeed);				//Home offset Speed
WriteUserParameterDINT(00,40,007,OffsetPosition);			//Home offset Position 
	
//40.009  AMC Home Maximum Allowed Move
//40.010  AMC Home Complete Window
WriteUserParameterDINT(00,40,009,MaxAllowedMove);			//Home Max Allowed Move
WriteUserParameterDINT(00,40,010,HomeCompleteWindow);		//Home Home Complete Window
	
//40.011  AMC Home On Freeze
//40.012  AMC Home Switch	
WriteUserParameterBOOL(00,40,011,TRUE);			//Home to Freeze
WriteUserParameterBOOL(00,40,013,FALSE);		//Stop now in the positive limit.  This are controlled by input 4 if bHomeNegativeDirection = FALSE
WriteUserParameterBOOL(00,40,014,FALSE);		//Stop now in the negative limit.  This are controlled by input 4 if bHomeNegativeDirection = True
			
WriteUserParameterBOOL(00,40,015,FALSE);		//40.015  AMC Home Positive Limit Selector
WriteUserParameterBOOL(00,40,016,FALSE);		//40.016  AMC Home Negative Limit Selector

WriteUserParameterLREAL(00,40,018,0);			//Torque level
WriteUserParameterLREAL(00,40,019,0);			//Torque Delay Time		

 
//Wait 4ms so the the Drive can see that the values changed.
Wait_Time(T#4MS);

	 
//Start the Homing using the trigger command and the normal command 
//34.007  AMC Reference Select
WriteUserParameterINT(00,34,007,5);					//5 = Start Homing

END_FUNCTION

// Drive/Application/Basic AMC Library/03 Commands/Home/Start_Homing_To_Torque
//Starts a home command that completes after a torque limit is reached for a given amount of time. 


//Version 0.00.03
//Cannon Melville 
FUNCTION Start_Homing_To_Torque
VAR_INPUT 
	Acceleration 		: DINT;
	Deceleration 		: DINT;
	Velocity			: DINT; 
	MaxAllowedMove		: DINT;	 // The max distance the home will run. 0 = disabled
	
	bHomeNegativeDirection	: BOOL;  // Home in the Negative Direction
	
	HomeCompleteWindow	: DINT;	 // This is used with the home complete flag
	HomeCompletePosition: DINT;  // This is the position of the homed after the torque value is reached.

	OffsetSpeed			: DINT;  // This is the speed the system will move as the position reset, after the home switch is found.
	OffsetPosition 		: DINT;  // This is the offset position from the home switch to go to after the home is done.
	
	TorqueThreshold		: LREAL; //Is the Torque percentage level needed to set home.
	TorqueTimeDelay		: LREAL; //How long the torque must be above the TorqueThreshold. Unit seconds with three decimal places.
	
	
	
END_VAR 
VAR

END_VAR

(*	 
	Editing the code in this function may result in limited support. 	 
*)

(*
	This block does not setup Input #4 for homing.
	if input #4 is mapped to home limit there will be a problem.
	so you might need to map 8.024 to 0 if it is mapped to menu 40
*)

(* NOTE
	Parameter 34.007  AMC Reference Select (Motion Commands)
	
	Value 	Disc 
	0 		Stop 
	1 		Position Abs 
	2 		Speed 
	3 		Cam 
	4 		EGB 
	5 		Home 
	6 		Position Rel 
	7 		Position Profile 
 
*)

//clear home offset 
WriteUserParameterDINT(00,33,003,0);						//clear position offset;
Wait_Time(T#30MS);											//wait 30 ms	


//Update profile generator 
//38.001  AMC Profile Acceleration
//38.002  AMC Profile Deceleration
//38.003  AMC Profile Maximum Speed
//40.003  AMC Home Maximum Speed
WriteUserParameterDINT(00,38,001,Acceleration);				//Set User Units Acceleration		UU/ ms^2
WriteUserParameterDINT(00,38,002,Deceleration);				//Set User Units Deceleration		UU/ ms^2
WriteUserParameterDINT(00,38,003,ABS(Velocity));			//Set User Units Velocity			UU/ ms
	

//menu 3
//03.100  F1 Freeze Trigger Source
//03.102  F1 Freeze Position Source
WriteUserParameterSINT(00,03,100,0);						//Use digital input 4
WriteUserParameterSINT(00,03,102,0);						//Use P1		
	
	
//menu 8
//WriteUserParameterLREAL(00,08,024,0); 						//map input 4 to nothing	
	
		
//Menu 40

//Direction settings
IF bHomeNegativeDirection THEN								//---- Negative direction ----	
	//40.002  AMC Home Mode
	WriteUserParameterSINT(00,40,002,3);					//Home mode 3  (i'm using this mode to do the neg direction)
	//40.013  AMC Home Positive Limit
	//40.014  AMC Home Negative Limit
	WriteUserParameterBOOL(00,40,015,FALSE);				//Disable the torque limit pos
	WriteUserParameterBOOL(00,40,016,TRUE);					//Enable the torque limit neg
 
	
	
ELSE														//---- Positive Direction ----
	//40.002  AMC Home Mode
	WriteUserParameterSINT(00,40,002,2);					//Home mode 2(i'm using this mode to do the Pos direction)
	//40.013  AMC Home Positive Limit
	//40.014  AMC Home Negative Limit
	WriteUserParameterBOOL(00,40,015,TRUE);					//Enable the torque limit pos
	WriteUserParameterBOOL(00,40,016,FALSE);				//Disable the torque limit neg 

END_IF



//40.001  AMC Home Direction
//40.003  AMC Home Maximum Speed
//40.004  AMC Home Position
WriteUserParameterBOOL(00,40,001,FALSE);					//Home Direction 
WriteUserParameterDINT(00,40,003,Velocity);					//Set User Units Velocity			UU/ms
WriteUserParameterDINT(00,40,004,HomeCompletePosition);		//Home  Switch Position
	 
//40.006  AMC Home Offset Maximum Speed
//40.007  AMC Home Offset Position
WriteUserParameterDINT(00,40,006,OffsetSpeed);				//Home offset Speed
WriteUserParameterDINT(00,40,007,OffsetPosition);			//Home offset Position 
	
//40.009  AMC Home Maximum Allowed Move
//40.010  AMC Home Complete Window
WriteUserParameterDINT(00,40,009,MaxAllowedMove);			//Home Max Allowed Move
WriteUserParameterDINT(00,40,010,HomeCompleteWindow);		//Home Home Complete Window
	
//40.011  AMC Home On Freeze
//40.012  AMC Home Switch	
WriteUserParameterBOOL(00,40,011,FALSE);					//dont use the freeze
WriteUserParameterBOOL(00,40,014,FALSE);					//Stop now limit.  Turn this off so the motion can run.
			
//40.015  AMC Home Positive Limit Selector
//40.016  AMC Home Negative Limit Selector
WriteUserParameterLREAL(00,40,018,TorqueThreshold);			//Torque level
WriteUserParameterLREAL(00,40,019,TorqueTimeDelay);			//Torque Delay Time		




//Wait 4ms so the the Drive can see that the values changed.
Wait_Time(T#4MS);

	 
//Start the Homing using the trigger command and the normal command 
//34.007  AMC Reference Select
WriteUserParameterINT(00,34,007,5);							//5 = Start Homing

END_FUNCTION

// Drive/Application/Basic AMC Library/03 Commands/Home/Start_Homing_To_Torque_Then_Input_4
//Starts a home command that completes after a torque limit is reached for a given amount of time. 


//Version 0.00.03
//Cannon Melville 
FUNCTION Start_Homing_To_Torque_Then_Input_4
VAR_INPUT 
	Acceleration 		: DINT;
	Deceleration 		: DINT;
	Velocity			: DINT; 
	MaxAllowedMove		: DINT;	 // The max distance the home will run. 0 = disabled
	
	bHomeNegativeDirection	: BOOL;  // Home in the Negative Direction
	
	HomeCompleteWindow	: DINT;	 // This is used with the home complete flag
	HomeCompletePosition: DINT;  // This is the position of the homed after the torque value is reached.

	OffsetSpeed			: DINT;  // This is the speed the system will move as the position reset, after the home switch is found.
	OffsetPosition 		: DINT;  // This is the offset position from the home switch to go to after the home is done.
	
	TorqueThreshold		: LREAL; //Is the Torque percentage level needed to set home.  Min = 0.1 max = 1000.0
	TorqueTimeDelay		: LREAL; //How long the torque must be above the TorqueThreshold. Unit seconds with three decimal places.
	bBackOffAfterTorque	: BOOL;  //after the torque Treshold and Torque Time Delay is met, Then reverse the directoin.
	
	
END_VAR 
VAR

END_VAR

(*	 
	Editing the code in this function may result in limited support. 	 
*)

(* NOTE
	Parameter 34.007  AMC Reference Select (Motion Commands)
	
	Value 	Disc 
	0 		Stop 
	1 		Position Abs 
	2 		Speed 
	3 		Cam 
	4 		EGB 
	5 		Home 
	6 		Position Rel 
	7 		Position Profile 
 
*)

//clear home offset
WriteUserParameterDINT(00,33,003,0);					//clear position offset;
Wait_Time(T#30MS);										//wait 30 ms	


//Update profile generator 
//38.001  AMC Profile Acceleration
//38.002  AMC Profile Deceleration
//38.003  AMC Profile Maximum Speed
//40.003  AMC Home Maximum Speed
WriteUserParameterDINT(00,38,001,Acceleration);				//Set User Units Acceleration		UU/ ms^2
WriteUserParameterDINT(00,38,002,Deceleration);				//Set User Units Deceleration		UU/ ms^2
WriteUserParameterDINT(00,38,003,ABS(Velocity));			//Set User Units Velocity			UU/ ms
	

//menu 3
//03.100  F1 Freeze Trigger Source
//03.102  F1 Freeze Position Source
WriteUserParameterSINT(00,03,100,0);						//Use digital input 4
WriteUserParameterSINT(00,03,102,0);						//Use P1		
	
	
//menu 8
WriteUserParameterLREAL(00,08,024,0); 						//map input 4 to nothing	
	

//menu 33 Slave freeze Select
//33.007  AMC Slave Freeze Select
WriteUserParameterBOOL(00,33,007,0);						//Select Freeze 1 input as home switch
	
		
//Menu 40

//Direction settings
IF bHomeNegativeDirection THEN								//---- Negative direction ----	
	//40.002  AMC Home Mode
	WriteUserParameterSINT(00,40,002,3);					//Home mode 3  (i'm using this mode to do the neg direction)
	//40.013  AMC Home Positive Limit
	//40.014  AMC Home Negative Limit
	WriteUserParameterBOOL(00,40,015,FALSE);				//Disable the torque limit pos
	WriteUserParameterBOOL(00,40,016,TRUE);					//Enable the torque limit neg
 
	 
	//40.001  AMC Home Direction after torque is met
	IF bBackOffAfterTorque THEN
		WriteUserParameterBOOL(00,40,001,FALSE);					//Home Direction 
	ELSE
		WriteUserParameterBOOL(00,40,001,TRUE);				//Home Direction 
	END_IF
	
ELSE														//---- Positive Direction ----
	//40.002  AMC Home Mode
	WriteUserParameterSINT(00,40,002,2);					//Home mode 2(i'm using this mode to do the Pos direction)
	//40.013  AMC Home Positive Limit
	//40.014  AMC Home Negative Limit
	WriteUserParameterBOOL(00,40,015,TRUE);					//Enable the torque limit pos
	WriteUserParameterBOOL(00,40,016,FALSE);				//Disable the torque limit neg 
 
	
	//40.001  AMC Home Direction after torque is met
	IF bBackOffAfterTorque THEN
		WriteUserParameterBOOL(00,40,001,TRUE);					//Home Direction 
	ELSE
		WriteUserParameterBOOL(00,40,001,FALSE);				//Home Direction 
	END_IF
	
END_IF



//40.003  AMC Home Maximum Speed
//40.004  AMC Home Position
WriteUserParameterDINT(00,40,003,Velocity);					//Set User Units Velocity			UU/ms
WriteUserParameterDINT(00,40,004,HomeCompletePosition);		//Home  Switch Position
	 
//40.006  AMC Home Offset Maximum Speed
//40.007  AMC Home Offset Position
WriteUserParameterDINT(00,40,006,OffsetSpeed);				//Home offset Speed
WriteUserParameterDINT(00,40,007,OffsetPosition);			//Home offset Position 
	
//40.009  AMC Home Maximum Allowed Move
//40.010  AMC Home Complete Window
WriteUserParameterDINT(00,40,009,MaxAllowedMove);			//Home Max Allowed Move
WriteUserParameterDINT(00,40,010,HomeCompleteWindow);		//Home Home Complete Window
	
//40.011  AMC Home On Freeze
//40.012  AMC Home Switch	
WriteUserParameterBOOL(00,40,011,TRUE);						//Home to Freeze
WriteUserParameterBOOL(00,40,014,FALSE);					//Stop now limit.  Turn this off so the motion can run.
			
//40.015  AMC Home Positive Limit Selector
//40.016  AMC Home Negative Limit Selector
WriteUserParameterLREAL(00,40,018,TorqueThreshold);			//Torque level
WriteUserParameterLREAL(00,40,019,TorqueTimeDelay);			//Torque Delay Time		




//Wait 4ms so the the Drive can see that the values changed.
Wait_Time(T#4MS);

	 
//Start the Homing using the trigger command and the normal command 
//34.007  AMC Reference Select
WriteUserParameterINT(00,34,007,5);							//5 = Start Homing

END_FUNCTION

// Drive/Application/Basic AMC Library/03 Commands/Home/Start_Homing_To_Torque_Then_Marker
//Starts a home command that completes after a torque limit is reached for a given amount of time. 


//Version 0.00.03
//Cannon Melville 
FUNCTION Start_Homing_To_Torque_Then_Marker
VAR_INPUT 
	Acceleration 		: DINT;
	Deceleration 		: DINT;
	Velocity			: DINT; 
	MaxAllowedMove		: DINT;	 // The max distance the home will run. 0 = disabled
	
	bHomeNegativeDirection	: BOOL;  // Home in the Negative Direction
	
	HomeCompleteWindow	: DINT;	 // This is used with the home complete flag
	HomeCompletePosition: DINT;  // This is the position of the homed after the torque value is reached.

	OffsetSpeed			: DINT;  // This is the speed the system will move as the position reset, after the home switch is found.
	OffsetPosition 		: DINT;  // This is the offset position from the home switch to go to after the home is done.
	
	TorqueThreshold		: LREAL; //Is the Torque percentage level needed to set home. Min = 0.1 max = 1000.0
	TorqueTimeDelay		: LREAL; //How long the torque must be above the TorqueThreshold. Unit seconds with three decimal places.
	bBackOffAfterTorque	: BOOL;  //after the torque Treshold and Torque Time Delay is met, Then reverse the directoin.

	
	
END_VAR 
VAR
 
END_VAR

(*	 
	Editing the code in this function may result in limited support. 	 
*)

(* NOTE
	Parameter 34.007  AMC Reference Select (Motion Commands)
	
	Value 	Disc 
	0 		Stop 
	1 		Position Abs 
	2 		Speed 
	3 		Cam 
	4 		EGB 
	5 		Home 
	6 		Position Rel 
	7 		Position Profile 
 
*)

//clear home offset
WriteUserParameterDINT(00,33,003,0);					//clear position offset;
Wait_Time(T#30MS);										//wait 30 ms	


//Update profile generator 
//38.001  AMC Profile Acceleration
//38.002  AMC Profile Deceleration
//38.003  AMC Profile Maximum Speed
//40.003  AMC Home Maximum Speed
WriteUserParameterDINT(00,38,001,Acceleration);				//Set User Units Acceleration		UU/ ms^2
WriteUserParameterDINT(00,38,002,Deceleration);				//Set User Units Deceleration		UU/ ms^2
WriteUserParameterDINT(00,38,003,ABS(Velocity));			//Set User Units Velocity			UU/ ms
	

//menu 3
//03.100  F1 Freeze Trigger Source
//03.102  F1 Freeze Position Source
IF ReadUserParameterSINT(00,03,038) = 0 OR ReadUserParameterSINT(00,03,038) = 3  THEN				//P1 Device Type(03.038) = AB Encoder then use marker else use 0 position Crossing
	WriteUserParameterSINT(00,03,100,2);					//Use digital P1 Marker
ELSE
	WriteUserParameterSINT(00,03,100,5);					//Use digital P1 Zero Position	
END_IF
WriteUserParameterSINT(00,03,102,0);						//Use P1		
	
	
//menu 8
WriteUserParameterLREAL(00,08,024,0); 						//map input 4 to nothing	
	

//menu 33 Slave freeze Select
//33.007  AMC Slave Freeze Select
WriteUserParameterBOOL(00,33,007,0);						//Select Freeze 1 input as home switch
	
	
		
//Menu 40

//Direction settings
IF bHomeNegativeDirection THEN								//---- Negative direction ----	
	//40.002  AMC Home Mode
	WriteUserParameterSINT(00,40,002,3);					//Home mode 3  (i'm using this mode to do the neg direction)
	//40.013  AMC Home Positive Limit
	//40.014  AMC Home Negative Limit
	WriteUserParameterBOOL(00,40,015,FALSE);				//Disable the torque limit pos
	WriteUserParameterBOOL(00,40,016,TRUE);					//Enable the torque limit neg
  
	//40.001  AMC Home Direction after torque is met
	IF bBackOffAfterTorque THEN
		WriteUserParameterBOOL(00,40,001,FALSE);					//Home Direction 
	ELSE
		WriteUserParameterBOOL(00,40,001,TRUE);				//Home Direction 
	END_IF
	
ELSE														//---- Positive Direction ----
	//40.002  AMC Home Mode
	WriteUserParameterSINT(00,40,002,2);					//Home mode 2(i'm using this mode to do the Pos direction)
	//40.013  AMC Home Positive Limit
	//40.014  AMC Home Negative Limit
	WriteUserParameterBOOL(00,40,015,TRUE);					//Enable the torque limit pos
	WriteUserParameterBOOL(00,40,016,FALSE);				//Disable the torque limit neg 

	
	//40.001  AMC Home Direction after torque is met
	IF bBackOffAfterTorque THEN
		WriteUserParameterBOOL(00,40,001,TRUE);					//Home Direction 
	ELSE
		WriteUserParameterBOOL(00,40,001,FALSE);				//Home Direction 
	END_IF
	
END_IF



//40.001  AMC Home Direction
//40.003  AMC Home Maximum Speed
//40.004  AMC Home Position
//WriteUserParameterBOOL(00,40,001,FALSE);					//Home Direction // Bug
WriteUserParameterDINT(00,40,003,Velocity);					//Set User Units Velocity			UU/ms
WriteUserParameterDINT(00,40,004,HomeCompletePosition);		//Home  Switch Position
	 
//40.006  AMC Home Offset Maximum Speed
//40.007  AMC Home Offset Position
WriteUserParameterDINT(00,40,006,OffsetSpeed);				//Home offset Speed
WriteUserParameterDINT(00,40,007,OffsetPosition);			//Home offset Position 
	
//40.009  AMC Home Maximum Allowed Move
//40.010  AMC Home Complete Window
WriteUserParameterDINT(00,40,009,MaxAllowedMove);			//Home Max Allowed Move
WriteUserParameterDINT(00,40,010,HomeCompleteWindow);		//Home Home Complete Window
	
//40.011  AMC Home On Freeze
//40.012  AMC Home Switch	
WriteUserParameterBOOL(00,40,011,TRUE);						//Home to Freeze
WriteUserParameterBOOL(00,40,014,FALSE);					//Stop now limit.  Turn this off so the motion can run.
			
//40.015  AMC Home Positive Limit Selector
//40.016  AMC Home Negative Limit Selector
WriteUserParameterLREAL(00,40,018,TorqueThreshold);			//Torque level
WriteUserParameterLREAL(00,40,019,TorqueTimeDelay);			//Torque Delay Time		




//Wait 4ms so the the Drive can see that the values changed.
Wait_Time(T#4MS);

	 
//Start the Homing using the trigger command and the normal command 
//34.007  AMC Reference Select
WriteUserParameterINT(00,34,007,5);							//5 = Start Homing

END_FUNCTION
